Staubli VAL3: description.pgx

program description(bool& x_bOk[])
  local num l_nI
  local num l_nWhich
begin
  //-----------------------------------------------------------------------
  //Header begin
  //Description of program
  //  This program lets you choose the keys to display
  //
  //Input parameters
  //  bool x_bOK
  //    role : User's choice: continue or stop the program
  //    possible values : 0 or 1 : 0 => Stop program, 1 => continue
  //
  //Traceability
  //  Creation : 07-04-08 - f.Rob
  //Header end
  //-----------------------------------------------------------------------

  x_bOk=false
  userPage()
  gotoxy(0,1)
  //Displays user instructions depending on the language defined
  for l_nI=(1+nLangSet) to (8+nLangSet)
    putln(sUsrMess[l_nI])
  endFor
  gotoxy(8,10)
  put(sUsrMess[23+nLangSet])
  //Functions to display navigation keys (F1 through F8)(here F3 and F6 with messages "YES" or "NO")
  call usrButtonTxt(3,sUsrMess[24+nLangSet])
  call usrButtonTxt(6,sUsrMess[25+nLangSet])
  //Waiting user choice: F3 or F6
  //F3=3 The user wants to continue
  //F6=6 The user wants to quit
  do
    l_nWhich=(get()-270)
  until ((l_nWhich==3) or (l_nWhich==6))
  //if the user wants to continue (he press F3) x_bOk passes true
  if l_nWhich==3
    x_bOk=true
  endIf
end
